Staubli VAL3: setLimit.pgx

program setLimit()
  local bool l_bRes
begin
  //set arm/cell limit:
  //
  l_bRes=$setArmLimits(jArmLimit[0],jArmLimit[1])
  if l_bRes
    gotoxy(1,11)
    put("setArmLimit:OK")
  else
    gotoxy(1,11)
    put("setArmLimit:fail")
  endIf
  //
  l_bRes=$setArmLimits(jCellLimit[0],jCellLimit[1])
  if l_bRes
    gotoxy(20,11)
    put("setCellLimit:OK")
  else
    gotoxy(20,11)
    put("setCellLimit:fail")
  endIf
end
